{attribute addProperty BoxType "EL2595-0000-0018"}
{attribute addProperty Id "DOX_StatusAT %I*DOX_Status_249B5F1F1620DOX_ControlAT %Q*DOX_Control_4111B8D51620WcStateAT %I*WcState_F855686C1620InfoDataAT %I*InfoData_BC63D37F80100"}
{attribute addProperty CRC "2948238325"}
{attribute addProperty SizeInBites "128"}
{attribute addProperty SizeInBytes "16"}
TYPE EL2595_74C0529E :
STRUCT
	{attribute addProperty Name "DOX_Status"}
	DOX_Status : DOX_Status_249B5F1F;
	{attribute addProperty Name "DOX_Control"}
	DOX_Control : DOX_Control_4111B8D5;
	{attribute addProperty Name "WcState"}
	WcState : WcState_F855686C;
	{attribute addProperty Name "InfoData"}
	InfoData : InfoData_BC63D37F;
END_STRUCT
END_TYPE

(* stored: Version 1.2.0.0, ProductVersion 3.1.4024.9
   DUT EL2595_74C0529E: Id {dbf2e45d-3aff-4916-9eba-c12178c8f30c} *)
